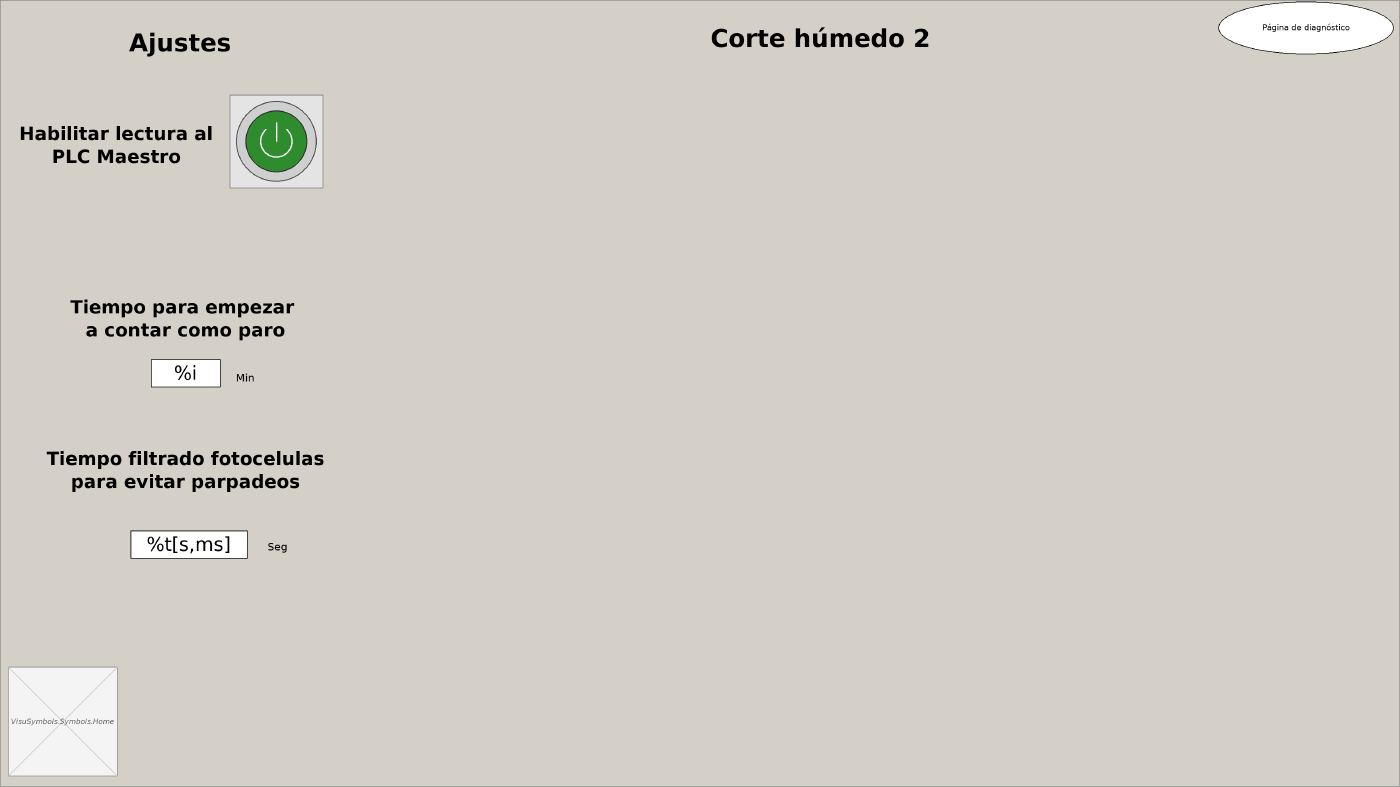
VISUALIZATION Ajustes_CorteH2  // 1920x1080
    Label (143,29 208x59), "Ajustes"
    Image (11,915 150x150), image: VisuSymbols.Symbols.Home
        OnMouseClick: change screen: Home_CortH2
    Label (22,144 275x110), "Habilitar lectura al PLC Maestro"
    PowerSwitch (315,128 128x132), variable: MAIN_Orden_Lectura_PLCs.bHabilitaLectura_Maestro, behaviour: TOGGLE, style: Switch-PowerSwitch-Green
    Label (82,390 345x94), "Tiempo para empezar a contar como paro"
    Label (160,482 188x30)
    Rectangle (207,493 95x38), "%i", text variable: FuncParoNodoRemote1CorteH2.HMI_Tiempo_Offset_MParo
        OnMouseDown: write the text variable via Edit
    Label (307,500 59x37), "Min"
    Label (58,598 393x94), "Tiempo filtrado fotocelulas para evitar parpadeos"
    Label (351,732 59x37), "Seg"
    Rectangle (179,728 160x38), "%t[s,ms]", text variable: FuncParoNodoRemote1CorteH2.HMI_TiempoFiltradoFotocel
        OnMouseDown: write the text variable via Edit
    Label (925,23 401x59), "Corte húmedo 2"
    Ellipse (1671,2 240x72), "Página de diagnóstico"
        OnMouseClick: change screen: DiagnosticoFB
END_VISUALIZATION

(* stored: Version 1.1.0.1, ProductVersion 3.1.4024.12
   Visu Ajustes_CorteH2: Id {5392cb0c-b2d1-4ac0-a9c2-16b7b91579bc} *)
